Staubli VAL3: stop.pgx

program stop()
  local string key
begin
  key = first(TASK_NAMES)

  while key != ""
    taskKill(TASK_NAMES[key])
    key = next(TASK_NAMES[key])
  endWhile

  disablePower()
end
